{attribute 'GeneratedUsingTerminal: EL4004-0000-0020'}
{attribute addProperty BoxType "EL4004-0000-0020"}
{attribute addProperty Id "Analog_outputAT %Q*INT2"}
{attribute addProperty CRC "3128867708"}
{attribute addProperty Size "2"}
TYPE AO_Outputs_Channel_BA7EBB7C :
STRUCT
	{attribute addProperty Name "Analog_output"}
	Analog_output AT %Q* : INT;
END_STRUCT
END_TYPE

(* stored: Version 1.2.0.0, ProductVersion 3.1.4024.9
   DUT AO_Outputs_Channel_BA7EBB7C: Id {a37604e5-f3f9-09db-06eb-5bc486a1e346} *)
